FUNCTION_BLOCK FB_MotionInterlocksCommon_Test EXTENDS FB_TestSuite
VAR
    fbMotionLogger 		: ARRAY[1..5] OF FB_MotionLogger;
END_VAR

GivenEpicsEnableAndHardwareEnableIfNotUserEnableThenResetPowerEnableAndMoveOk_Test1();
GivenEpicsEnablehardwareEnableAndUserEnableUpdatePowerEnableAndMoveOk_Test2();
GivenhardwareEnableAndUserEnableIfNotEpicsEnableResetPowerEnable_Test3();
GivenUserEnableAndDriveEnableIfNothardwareEnableThenTriggerHardwareEnableInterlockAndRemoveMoveOk_Test4();
GivenInterlockEventIFGlobalResetClearErrors_Test5();

METHOD PRIVATE GivenEpicsEnableAndHardwareEnableIfNotUserEnableThenResetPowerEnableAndMoveOk_Test1
VAR
    fbMotionInterlocksCommon : FB_MotionInterlocksCommon(iMotionLogger:=fbMotionLogger[1]);
    sExpectedUserEnableMessage : STRING := 'User enable interlock triggered!';
    sActUserEnableMessage : STRING;
END_VAR
TEST(__POUNAME());
// Test UserEnable interlock trigger
fbMotionInterlocksCommon.HardwareEnable := TRUE;
fbMotionInterlocksCommon.UserEnable := FALSE;
fbMotionInterlocksCommon.DriveCommands(Enable:=TRUE, NewMoveReq:=FALSE);
fbMotionInterlocksCommon();

AssertFalse(Condition := fbMotionInterlocksCommon.PowerEnabled,
           Message := 'UserEnbale Interlock triggered PowerEnable must be unset #1');

AssertFalse(Condition := fbMotionInterlocksCommon.MoveOk,
           Message := 'UserEnbale Interlock triggered MoveOk must be unset #2');

sActUserEnableMessage := fbMotionInterlocksCommon.Message;
AssertEquals ( Expected:=sExpectedUserEnableMessage, Actual:=sActUserEnableMessage,
            Message:='Incorrect UserEnbale trigger Error Msg #3');

TEST_FINISHED();
END_METHOD

METHOD PRIVATE GivenEpicsEnablehardwareEnableAndUserEnableUpdatePowerEnableAndMoveOk_Test2
VAR
    fbMotionInterlocksCommon : FB_MotionInterlocksCommon(iMotionLogger:=fbMotionLogger[2]);
    sExpectedMessage : STRING := '';
    sActMessage : STRING;
    nExpectedErrorId : UDINT := 0;
    nActErrorId : UDINT;
END_VAR
TEST(__POUNAME());
// PowerEnable and MoveOk Set
fbMotionInterlocksCommon.HardwareEnable := TRUE;
fbMotionInterlocksCommon.UserEnable := TRUE;
fbMotionInterlocksCommon.DriveCommands(Enable:=TRUE, NewMoveReq:=FALSE);
fbMotionInterlocksCommon();

AssertTrue(Condition := fbMotionInterlocksCommon.PowerEnabled,
           Message := 'Hardware or UserEnable Interlock not set #1');

AssertTrue(Condition := fbMotionInterlocksCommon.MoveOk,
           Message := 'Hardware or UserEnable Interlock not set #2');

AssertFalse(Condition := fbMotionInterlocksCommon.Error,
           Message := 'No Error expected #3');

nActErrorId := fbMotionInterlocksCommon.ErrorID;
AssertEquals ( Expected:=nExpectedErrorId, Actual:=nActErrorId ,
            Message:='ErrorID must be 0 #4');

sActMessage := fbMotionInterlocksCommon.Message;
AssertEquals ( Expected:=sExpectedMessage, Actual:=sActMessage ,
            Message:='No error Message #5');

TEST_FINISHED();
END_METHOD

METHOD PRIVATE GivenhardwareEnableAndUserEnableIfNotEpicsEnableResetPowerEnable_Test3
VAR
    fbMotionInterlocksCommon : FB_MotionInterlocksCommon(iMotionLogger:=fbMotionLogger[3]);
    sExpectedMessage : STRING := '';
    sActMessage : STRING;
    nExpectedErrorId : UDINT := 0;
    nActErrorId : UDINT;
END_VAR
TEST(__POUNAME());
// EpicsEnable Interlock trigger
fbMotionInterlocksCommon.HardwareEnable := TRUE;
fbMotionInterlocksCommon.UserEnable := TRUE;

fbMotionInterlocksCommon.DriveCommands(Enable:=FALSE, NewMoveReq:=FALSE);
fbMotionInterlocksCommon();

AssertFalse(Condition := fbMotionInterlocksCommon.PowerEnabled,
           Message := 'No Epics Enable, PowerEnabled must not be set #1');

AssertTrue(Condition := fbMotionInterlocksCommon.MoveOk,
           Message := 'Epics Enable reset, Move Request must be invalid #2');

AssertFalse(Condition := fbMotionInterlocksCommon.Error,
           Message := 'No Error expected #3');

nActErrorId := fbMotionInterlocksCommon.ErrorID;
AssertEquals ( Expected:=nExpectedErrorId, Actual:=nActErrorId ,
            Message:='ErrorID must be 0 #4');

sActMessage := fbMotionInterlocksCommon.Message;
AssertEquals ( Expected:=sExpectedMessage, Actual:=sActMessage ,
            Message:='No error Message #5');
TEST_FINISHED();
END_METHOD

METHOD PRIVATE GivenInterlockEventIFGlobalResetClearErrors_Test5
VAR
    fbMotionInterlocksCommon : FB_MotionInterlocksCommon(iMotionLogger:=fbMotionLogger[5]);
    sExpectedMessage : STRING := '';
    sActMessage : STRING;
    nExpectedErrorId : UDINT := 0;
    nActErrorId : UDINT;
END_VAR
TEST(__POUNAME());
// HardwareEnable unset
fbMotionInterlocksCommon.UserEnable := TRUE;
fbMotionInterlocksCommon.HardwareEnable := FALSE;
fbMotionInterlocksCommon.DriveCommands(Enable:=FALSE, NewMoveReq:=FALSE);
fbMotionInterlocksCommon();

AssertTRUE(Condition := fbMotionInterlocksCommon.Error,
           Message := 'HardwareEnable Error must be set #1');

// Test Global Reset to clear internal flags
fbMotionInterlocksCommon.HardwareEnable := TRUE;
fbMotionInterlocksCommon.Reset();
fbMotionInterlocksCommon();

AssertFalse(Condition := fbMotionInterlocksCommon.Error,
           Message := 'Error must be clear after global reset #2');

sActMessage := fbMotionInterlocksCommon.Message;
AssertEquals ( Expected:=sExpectedMessage, Actual:=sActMessage,
            Message:='Error Msg must be cleared #3');
TEST_FINISHED();
END_METHOD

METHOD PRIVATE GivenUserEnableAndDriveEnableIfNothardwareEnableThenTriggerHardwareEnableInterlockAndRemoveMoveOk_Test4
VAR
    fbMotionInterlocksCommon : FB_MotionInterlocksCommon(iMotionLogger:=fbMotionLogger[4]);
    sExpectedHardwareEnableMessage : STRING := 'Hardware enbale interlocks triggered!';
    sActHardwareEnableMessage : STRING;
    nExpectedErrorId : UDINT := 11;
    nActErrorId : UDINT;
END_VAR
TEST(__POUNAME());
// HardwareEnable unset
fbMotionInterlocksCommon.UserEnable := TRUE;
fbMotionInterlocksCommon.HardwareEnable := FALSE;
fbMotionInterlocksCommon.DriveCommands(Enable:=TRUE, NewMoveReq:=FALSE);
fbMotionInterlocksCommon();

AssertFalse(Condition := fbMotionInterlocksCommon.PowerEnabled,
           Message := 'Hardware Interlock triggered PowerEnable must be unset #1');

AssertFalse(Condition := fbMotionInterlocksCommon.MoveOk,
           Message := 'Hardware Interlock triggered MoveOk must be unset #2');

AssertTrue(Condition := fbMotionInterlocksCommon.Error,
           Message := 'Hardware Interlock triggered Error must be set #3');

nActErrorId := fbMotionInterlocksCommon.ErrorID;
AssertEquals ( Expected:=nExpectedErrorId, Actual:=nActErrorId , Message:='Incorrect Hardware trigger ErrorID #4');

sActHardwareEnableMessage := fbMotionInterlocksCommon.Message;
AssertEquals ( Expected:=sExpectedHardwareEnableMessage, Actual:=sActHardwareEnableMessage , Message:='Incorrect Hardware trigger Error Msg #5');

TEST_FINISHED();
END_METHOD

END_FUNCTION_BLOCK

(* stored: Version 1.1.0.1
   POU FB_MotionInterlocksCommon_Test: Id {a2005ca9-592c-499d-b205-56dd47273a45}, SpecialFunc None
   Method GivenEpicsEnableAndHardwareEnableIfNotUserEnableThenResetPowerEnableAndMoveOk_Test1: Id {2fccb30b-fa43-4cab-8f2c-adfb09669aa8}
   Method GivenEpicsEnablehardwareEnableAndUserEnableUpdatePowerEnableAndMoveOk_Test2: Id {29a6cbb8-e701-4efa-8b8e-943b61227a98}
   Method GivenhardwareEnableAndUserEnableIfNotEpicsEnableResetPowerEnable_Test3: Id {71eb458d-3e16-42c1-906d-1967152b9a7a}
   Method GivenInterlockEventIFGlobalResetClearErrors_Test5: Id {26b812f8-7691-4546-890b-17127a999f93}
   Method GivenUserEnableAndDriveEnableIfNothardwareEnableThenTriggerHardwareEnableInterlockAndRemoveMoveOk_Test4: Id {0b67d0e3-11d8-4176-a42c-58d4ebf9caa3} *)
